// Block: FlyingCarriage_PERS

DATA_BLOCK FlyingCarriage_PERS
VERSION : 0.1
   NON_RETAIN
   VAR
      Parameter : udt_FlyingCarriage_Parameter;
      FsParameter : udt_FsParameter;
      SLS_Vel : LReal;
   END_VAR

BEGIN
   // No initialization required
END_DATA_BLOCK
